(* CoDeSys 2.3.9.475 project: bmsProg.pro *)
(* Libraries: WagoCANLayer2_02.lib 23.6.14 12:08:28, Standard.lib 20.5.14 07:13:26, Iecsfc.lib 16.5.13 13:00:50, SYSLIBCALLBACK.LIB 16.5.13 13:00:50 *)

(* PLC configuration (modules and I/O channels)
K-Bus [K_Bus] node 0, in %IB0 out %QB0 {KbusBusMode = 1; KbusCycleTime = 10000; KbusThreadPriority = 0; KbusSetOutputsToZeroOnApplicationStop = 1}
Modbus variables [PFC200MODBUS] node 1, in %IB0 out %QB0 {PlcStopBehaviour = 1; FiledbusErrorBehaviour = 1; TcpOperation = 1; TcpPort = 502; TcpTimeout = 600; UdpOperation = 1; UdpPort = 502; RtuOperation = 0; NodeId = 1; ResponseTimeout = 5000; Interface = 0; Baud = 115200; StopBits = 1; Parity = 1; FlowCtrl = 0; PhysInterface = 0}
CAN Layer2 Device [PFC200CANLAYER2] node 2, in %IB6000 out %QB6000 {PFC200CanLayer2NONE = 0}
Modbus-Master [MB_MASTER] node 3, in %IB0 out %QB0
*)

(* Task configuration *)
TASK T100 (PRIORITY := 6, INTERVAL := T#1000ms);
	PLC_PRG();
END_TASK

(* POU PLC_PRG, ST *)
PROGRAM PLC_PRG
VAR
	xOpenPort			: BOOL;
	fbOpenPort		: CAN_OPEN;
	xPortIsOpen		: BOOL;

	fbCanSend305			: CAN_TX_11BIT_FRAME :=(
		CAN_ID			       := 16#305,
		RTR_FRAME		:= FALSE,
		DATALENGTH	:= 8 );
	fbCanSend306			: CAN_TX_11BIT_FRAME :=(
		CAN_ID			:= 16#306,
		RTR_FRAME		:= FALSE,
		DATALENGTH	:= 8 );
	fbCanSendRelay307	: CAN_TX_11BIT_FRAME :=(
		CAN_ID			:= 16#307,
		RTR_FRAME		:= FALSE,
		DATALENGTH	:= 8 );
	fbCanSendAlarmsBMS	: CAN_TX_11BIT_FRAME :=(
		CAN_ID				:= 16#35A,
		RTR_FRAME			:= FALSE,
		DATALENGTH	:= 8 );
	fbCanSend355 	: CAN_TX_11BIT_FRAME :=(
		CAN_ID				:= 16#355,
		RTR_FRAME			:= FALSE,
		DATALENGTH	:= 8 );
	fbCanSend351 	: CAN_TX_11BIT_FRAME :=(
		CAN_ID				:= 16#351,
		RTR_FRAME			:= FALSE,
		DATALENGTH	:= 8 );
	fbCanSend356	: CAN_TX_11BIT_FRAME :=(
		CAN_ID				:= 16#356,
		RTR_FRAME			:= FALSE,
		DATALENGTH	:= 8 );


	fbCanRecvBMS355	 : CAN_RX_11BIT_FRAME :=	(
		CAN_ID 			:= 16#355,
		CAN_BUFFER	:= FALSE );
	fbCanRecvBMS351	 : CAN_RX_11BIT_FRAME :=	(
		CAN_ID 			:= 16#351,
		CAN_BUFFER	:= FALSE );
	fbCanRecvBMS356 : CAN_RX_11BIT_FRAME :=	(
		CAN_ID 			:= 16#356,
		CAN_BUFFER	:= FALSE );
	fbCanRecv305			: CAN_RX_11BIT_FRAME :=(
		CAN_ID			:= 16#305,
		CAN_BUFFER	:= FALSE );
	fbCanRecv306			: CAN_RX_11BIT_FRAME :=(
	CAN_ID			:= 16#306,
		CAN_BUFFER	:= FALSE );
	fbCanRecv307			: CAN_RX_11BIT_FRAME :=(
		CAN_ID			:= 16#307,
		CAN_BUFFER	:= FALSE );

	xWrite					: BOOL;
	xRead					: BOOL;
	wState					: WORD;

	aSendData305			: ARRAY [1..8] OF BYTE :=3,2,1,0,196,0,14,1;
	aSendData306			: ARRAY [1..8] OF BYTE := 100,0,10,1,0,0,93,2;
	aSendData307			: ARRAY [1..8] OF BYTE :=  62,6,64,49,62,6,64,49;
	aSendData35A			: ARRAY [1..8] OF BYTE  := 170, 170, 170, 170, 170, 170, 170,  170; (*Alarm/Warning external BMS*)
	aSendData351			: ARRAY [1..8] OF BYTE := 103,2,52,3,126,9,164,1;
	aSendData355			: ARRAY [1..8] OF BYTE := 27,0,100,0,140,10,0,0;
	aSendData356 			: ARRAY[1..8] OF BYTE := 50,20,255,255,196,0,0,0;


	aRecvData305			: ARRAY [1..8] OF BYTE;
	aRecvData306			: ARRAY [1..8] OF BYTE;
	socRev355			       : ARRAY [1..8] OF BYTE;
	btV351 					: ARRAY [1..8] OF BYTE;
	(*bRecvLen				: BYTE;*)
	tSend						: TON :=(PT:= t#300ms );
END_VAR
fbOpenPort(BAUDRATE:= 500000, ENABLE:= xOpenPort);

fbCanRecv305(
	ENABLE:= xPortIsOpen,
	READ_FRAME:= xRead );
fbCanRecv306(
	ENABLE:= xPortIsOpen,
	READ_FRAME:= xRead );
fbCanRecv307(
	ENABLE:= xPortIsOpen,
	READ_FRAME:= xRead );
fbCanRecvBMS355(
	ENABLE:= xPortIsOpen,
	READ_FRAME:= xRead );
fbCanRecvBMS351(
	ENABLE:= xPortIsOpen,
	READ_FRAME:= xRead );
fbCanRecvBMS356(
	ENABLE:= xPortIsOpen,
	READ_FRAME:= xRead );

(*timeout sunny island *)
fbCanSend355(
	DATA:= aSendData355,
	ENABLE:= xPortIsOpen,
	WRITE_FRAME:= xWrite
);
fbCanSend351(
	DATA:= aSendData351,
	ENABLE:= xPortIsOpen,
	WRITE_FRAME:= xWrite
);
fbCanSend356(
	DATA:= aSendData356,
	ENABLE:= xPortIsOpen,
	WRITE_FRAME:= xWrite
);
fbCanSendAlarmsBMS(
	DATA:= aSendData35A,
	ENABLE:= xPortIsOpen,
	WRITE_FRAME:= xWrite );

fbCanSend305(
	DATA:= aSendData305,
	ENABLE:= xPortIsOpen,
	WRITE_FRAME:= xWrite );
fbCanSend306(
	DATA:= aSendData306,
	ENABLE:= xPortIsOpen,
	WRITE_FRAME:= xWrite );
fbCanSendRelay307(
	DATA:= aSendData307,
	ENABLE:= xPortIsOpen,
	WRITE_FRAME:= xWrite );


CASE wState OF
0: (* open CAN port *)
	xOpenPort := TRUE;
	IF fbOpenPort.CONFIRM AND fbOpenPort.ERROR = CAN_PORT_OK THEN
		xOpenPort := FALSE;
		xPortIsOpen := TRUE;
		wState := 10;
	END_IF
10: (* send cyclic messages and check if message was received *)
	tSend(IN := TRUE AND NOT xWrite);
	IF tSend.Q THEN (* sending message *)
		tSend(IN := FALSE);
		xWrite := TRUE;
	ELSIF NOT xRead THEN (* message received *)
		IF fbCanRecv305.ERROR = CAN_RECEIVE_OK OR  fbCanRecv306.ERROR = CAN_RECEIVE_OK
			OR  fbCanRecv307.ERROR = CAN_RECEIVE_OK OR fbCanRecvBMS355.ERROR = CAN_RECEIVE_OK
			OR fbCanRecvBMS351.ERROR = CAN_RECEIVE_OK THEN

			aRecvData305 := fbCanRecv305.DATA;
			aRecvData306 := fbCanRecv306.DATA;
			(*aRecvData3 := fbCanRecv307.DATA;*)
			socRev355 	:= fbCanRecvBMS355.DATA;
			btV351		  	:= fbCanRecvBMS351.DATA;

			(*16#305*)
			(*aSendData305[1] := aRecvData305[1]; (*nach ausschalten leer*)
			aSendData305[2] := aRecvData305[2];
			aSendData305[3] := aRecvData305[3];
			aSendData305[4] := aRecvData305[4];
			aSendData305[5] := aRecvData305[5];
			aSendData305[6] := aRecvData305[6];
			aSendData305[7] := socRev355[1]; (*SOC*)
			aSendData305[8] := socRev355[2];*)

			(*16#306*)
			(*aSendData306[1] := socRev355[3]; (*SOH*)
			aSendData306[2] := socRev355[4];
			aSendData306[3] := 10;
			aSendData306[4] := 1;
			aSendData306[5] := 0;
			aSendData306[6] := 0;
			aSendData306[7] := btV351[1]; (*charging volate ?*)
			aSendData306[8] := btV351[2];*)

			(*FOR iVar_1 :=1 TO 10 BY 1 DO *)
			(*aSendData307			 :=  62,6,64,49,62,6,64,49 ;
			aSendData35A			 := 170, 170, 170, 170, 170, 170, 170,  170 ;*)

			(*bRecvLen := fbCanRecv1.DATALENGTH;*)
			xRead := TRUE;
		ELSE
			xRead := TRUE;
		END_IF
	END_IF
END_CASE
END_PROGRAM

(* POU Configuration/MODBUS_CONFIGURATION, ST *)
PROGRAM MODBUS_CONFIGURATION        
VAR                                
END_VAR                            
(*                                 
   <?xml version="1.0" encoding="UTF-16" standalone="yes"?>
<network xml_structure_version="1" xml_feature_version="1">
	<generator_settings minRTUTaskCycleTimeMs="5" minEthaskCycleTimeMs="5" ethSlaveMultiplier="0.1" rtuInterfaceMultiplier="0.1" taskGeneration="false"/>
</network>
                              
*)                                 
;                                  
END_PROGRAM
